(* Logix 5000 project; controller Receptivo vendor 1 type 14 code 106 rev 30.11; software revision 30.00; part 9 of 10 *)
(* tags used below, declared in another part *)
   Command_Status : DINT;
   Gway_Error : BOOL;
   GWay_Heartbeat : DINT;
   Gway_Status : DINT;
   ons_tare_station_3 : BOOL;
   ons_wpm3 : BOOL;
   ons_wpm4 : BOOL;
   Timer_Gway_Hearbeat : TIMER[4];
   Timer_Tare_Station_3 : TIMER;
   Timer_Tare_Station_3_aux : BOOL;
   Timer_Tare_Station_4 : TIMER;
   Timer_Tare_Station_4_aux : BOOL;
   Timer_WPM3_Heartbeat : TIMER[8];
   Timer_WPM4_Heartbeat : TIMER[8];
   WPM_3_COUNT_ANTERIOR : DINT;
   WPM_4_COUNT_ANTERIOR : DINT;
   ACTIVE_SLOT : DINT[10];
   CAJAS_1 : DINT;
   CAJAS_2 : DINT;
   CAJAS_3 : DINT;
   CAJAS_4 : DINT;
   CHASSIS_LAST : DINT;
   Diff_Peso_1 : DINT;
   Diff_Peso_2 : DINT;
   Diff_Peso_3 : DINT;
   Diff_Peso_4 : DINT;
   FORCE_STATUS : DINT;
   KEY_SWITCH_RUN : BOOL;
   MODULE_FAULT_STATUS : DINT[10];
   Num_Cajas_Reales_1 : DINT;
   Num_Cajas_Reales_2 : DINT;
   Num_Cajas_Reales_3 : DINT;
   Num_Cajas_Reales_4 : DINT;
   ons_tare_station_4 : BOOL;
   PB_Tare_Station_3 : BOOL;
   PB_Tare_Station_4 : BOOL;
   Peso_OK_Estacion_1 : BOOL;
   Peso_OK_Estacion_2 : BOOL;
   Peso_OK_Estacion_3 : BOOL;
   Peso_OK_Estacion_4 : BOOL;
   PESO_REAL_1 : DINT;
   PESO_REAL_2 : DINT;
   PESO_REAL_3 : DINT;
   PESO_REAL_4 : DINT;
   PESO_TEORICO_1 : DINT;
   PESO_TEORICO_2 : DINT;
   PESO_TEORICO_3 : DINT;
   PESO_TEORICO_4 : DINT;
   Porcentaje_Peso_1 : REAL;
   Porcentaje_Peso_2 : REAL;
   Porcentaje_Peso_3 : REAL;
   Porcentaje_Peso_4 : REAL;
   Producto1 : UDT_Inventario;
   Producto2 : UDT_Inventario;
   Producto3 : UDT_Inventario;
   Producto4 : UDT_Inventario;
   Station3_Tare_OK : BOOL;
   Station4_Tare_OK : BOOL;
   SYSTEM_ALARMS : DINT[10];
   Tara_1 : DINT;
   Tara_2 : DINT;
   Tara_3 : DINT;
   Tara_4 : DINT;
   Tara_Fecha_Estacion_3 : Hora_y_Fecha;
   Tara_Fecha_Estacion_4 : Hora_y_Fecha;
   Tare_Station_1_Write : DINT;
   Tare_Station_2_Write : DINT;
   Tare_Station_3_Write : DINT;
   Tare_Station_4_Write : DINT;
   WPM1_Heartbeat_Error : BOOL;
   WPM2_Heartbeat_Error : BOOL;
   WPM3_Heartbeat : DINT;
   WPM3_Heartbeat_Error : BOOL;
   WPM3_Status : WPM_Status;
   WPM4_Heartbeat : DINT;
   WPM4_Heartbeat_Error : BOOL;
   WPM4_Status : WPM_Status;
   WPM_3_Selected : DINT;
   WPM_3_Status_Aux : DINT;
   WPM_4_Selected : DINT;
   WPM_4_Status_Aux : DINT;
   Zero : DINT;
(* Pesaje, continued *)

ROUTINE Control_Pesaje_3   (* ladder *)
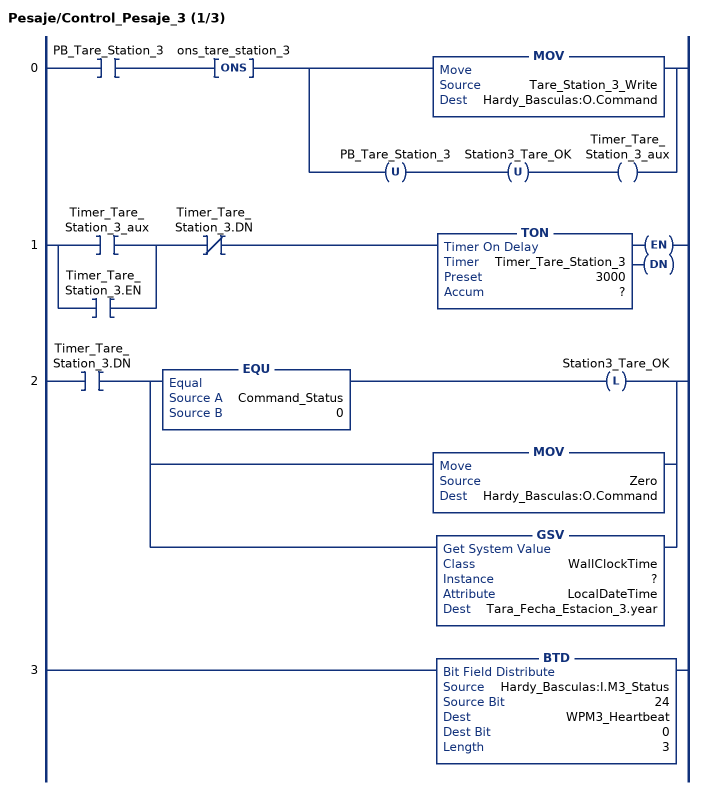
   0: XIC(PB_Tare_Station_3)ONS(ons_tare_station_3)[MOV(Tare_Station_3_Write,Hardy_Basculas:O.Command) ,OTU(PB_Tare_Station_3) OTU(Station3_Tare_OK) OTE(Timer_Tare_Station_3_aux) ];
   1: [XIC(Timer_Tare_Station_3_aux) ,XIC(Timer_Tare_Station_3.EN) ]XIO(Timer_Tare_Station_3.DN)TON(Timer_Tare_Station_3,?,?);
   2: XIC(Timer_Tare_Station_3.DN)[EQU(Command_Status,0) OTL(Station3_Tare_OK) ,MOV(Zero,Hardy_Basculas:O.Command) ,GSV(WallClockTime,?,LocalDateTime,Tara_Fecha_Estacion_3.year) ];
   3: BTD(Hardy_Basculas:I.M3_Status,24,WPM3_Heartbeat,0,3);
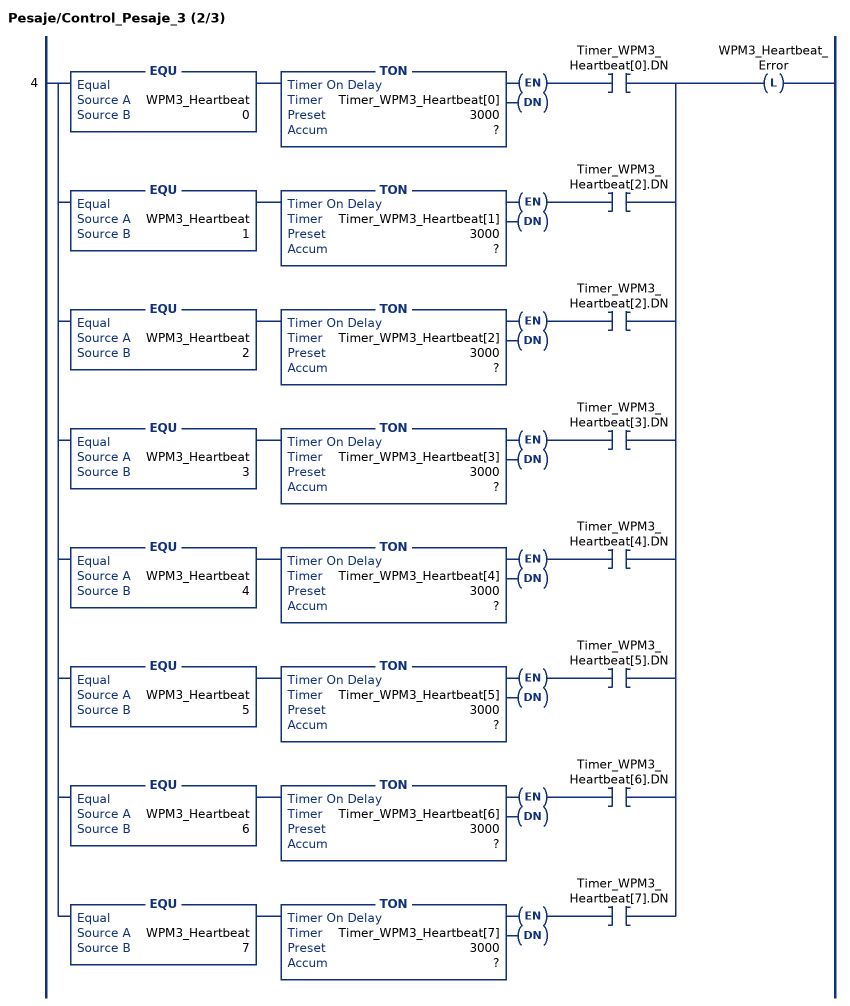
   4: [EQU(WPM3_Heartbeat,0) TON(Timer_WPM3_Heartbeat[0],?,?) XIC(Timer_WPM3_Heartbeat[0].DN) ,EQU(WPM3_Heartbeat,1) TON(Timer_WPM3_Heartbeat[1],?,?) XIC(Timer_WPM3_Heartbeat[2].DN) ,EQU(WPM3_Heartbeat,2) TON(Timer_WPM3_Heartbeat[2],?,?) XIC(Timer_WPM3_Heartbeat[2].DN) ,EQU(WPM3_Heartbeat,3) TON(Timer_WPM3_Heartbeat[3],?,?) XIC(Timer_WPM3_Heartbeat[3].DN) ,EQU(WPM3_Heartbeat,4) TON(Timer_WPM3_Heartbeat[4],?,?) XIC(Timer_WPM3_Heartbeat[4].DN) ,EQU(WPM3_Heartbeat,5) TON(Timer_WPM3_Heartbeat[5],?,?) XIC(Timer_WPM3_Heartbeat[5].DN) ,EQU(WPM3_Heartbeat,6) TON(Timer_WPM3_Heartbeat[6],?,?) XIC(Timer_WPM3_Heartbeat[6].DN) ,EQU(WPM3_Heartbeat,7) TON(Timer_WPM3_Heartbeat[7],?,?) XIC(Timer_WPM3_Heartbeat[7].DN) ]OTL(WPM3_Heartbeat_Error);
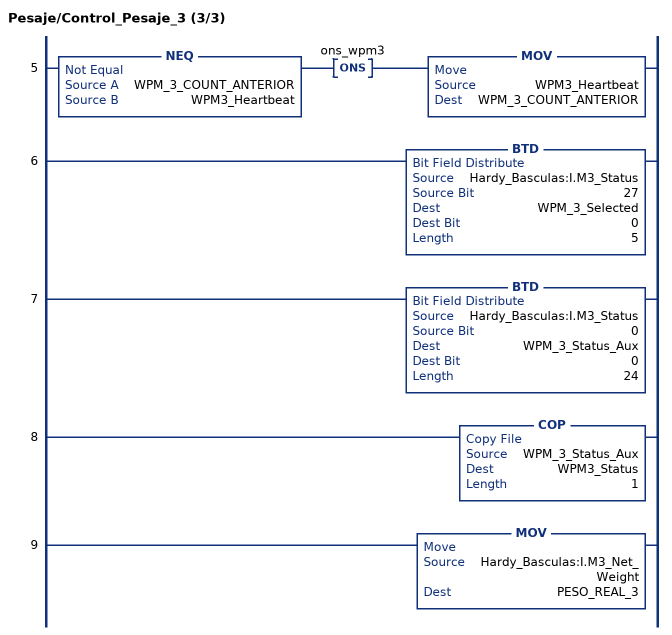
   5: NEQ(WPM_3_COUNT_ANTERIOR,WPM3_Heartbeat)ONS(ons_wpm3)MOV(WPM3_Heartbeat,WPM_3_COUNT_ANTERIOR);
   6: BTD(Hardy_Basculas:I.M3_Status,27,WPM_3_Selected,0,5);
   7: BTD(Hardy_Basculas:I.M3_Status,0,WPM_3_Status_Aux,0,24);
   8: COP(WPM_3_Status_Aux,WPM3_Status,1);
   9: MOV(Hardy_Basculas:I.M3_Net_Weight,PESO_REAL_3);
END_ROUTINE

ROUTINE Control_Pesaje_4   (* ladder *)
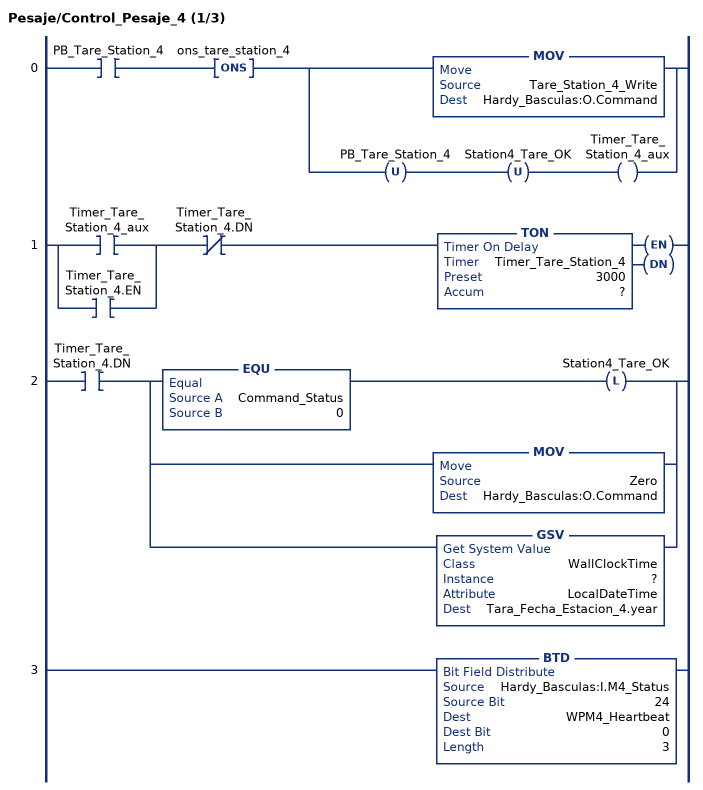
   0: XIC(PB_Tare_Station_4)ONS(ons_tare_station_4)[MOV(Tare_Station_4_Write,Hardy_Basculas:O.Command) ,OTU(PB_Tare_Station_4) OTU(Station4_Tare_OK) OTE(Timer_Tare_Station_4_aux) ];
   1: [XIC(Timer_Tare_Station_4_aux) ,XIC(Timer_Tare_Station_4.EN) ]XIO(Timer_Tare_Station_4.DN)TON(Timer_Tare_Station_4,?,?);
   2: XIC(Timer_Tare_Station_4.DN)[EQU(Command_Status,0) OTL(Station4_Tare_OK) ,MOV(Zero,Hardy_Basculas:O.Command) ,GSV(WallClockTime,?,LocalDateTime,Tara_Fecha_Estacion_4.year) ];
   3: BTD(Hardy_Basculas:I.M4_Status,24,WPM4_Heartbeat,0,3);
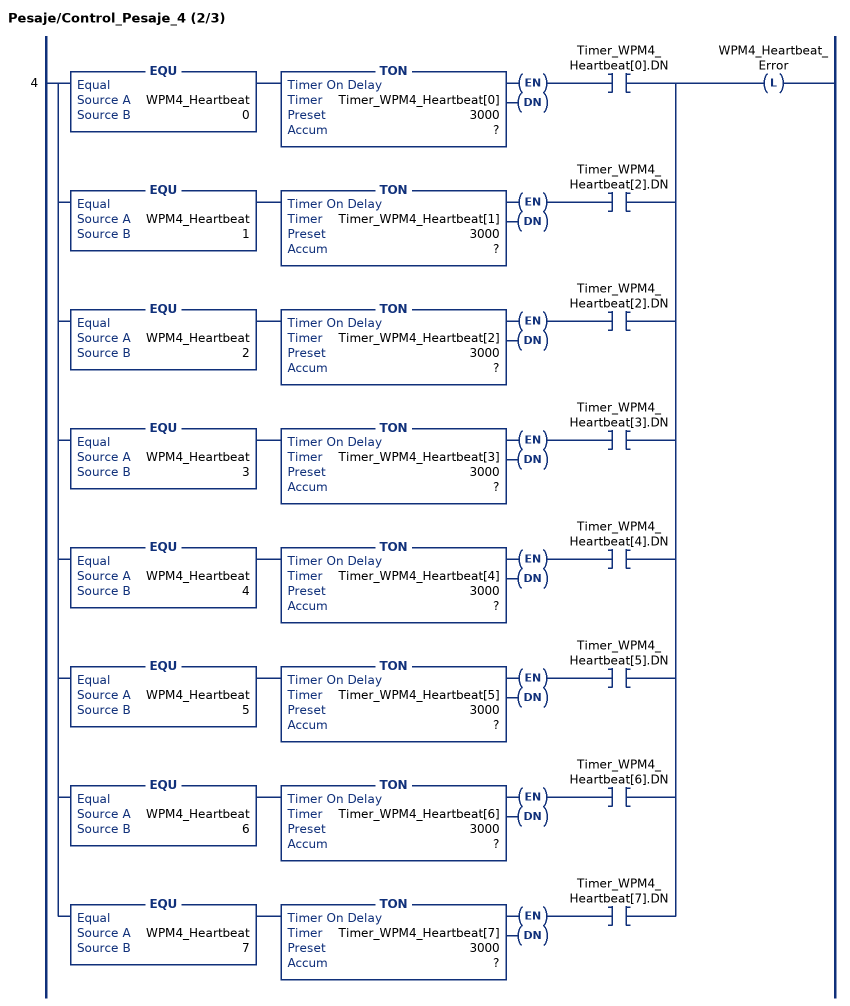
   4: [EQU(WPM4_Heartbeat,0) TON(Timer_WPM4_Heartbeat[0],?,?) XIC(Timer_WPM4_Heartbeat[0].DN) ,EQU(WPM4_Heartbeat,1) TON(Timer_WPM4_Heartbeat[1],?,?) XIC(Timer_WPM4_Heartbeat[2].DN) ,EQU(WPM4_Heartbeat,2) TON(Timer_WPM4_Heartbeat[2],?,?) XIC(Timer_WPM4_Heartbeat[2].DN) ,EQU(WPM4_Heartbeat,3) TON(Timer_WPM4_Heartbeat[3],?,?) XIC(Timer_WPM4_Heartbeat[3].DN) ,EQU(WPM4_Heartbeat,4) TON(Timer_WPM4_Heartbeat[4],?,?) XIC(Timer_WPM4_Heartbeat[4].DN) ,EQU(WPM4_Heartbeat,5) TON(Timer_WPM4_Heartbeat[5],?,?) XIC(Timer_WPM4_Heartbeat[5].DN) ,EQU(WPM4_Heartbeat,6) TON(Timer_WPM4_Heartbeat[6],?,?) XIC(Timer_WPM4_Heartbeat[6].DN) ,EQU(WPM4_Heartbeat,7) TON(Timer_WPM4_Heartbeat[7],?,?) XIC(Timer_WPM4_Heartbeat[7].DN) ]OTL(WPM4_Heartbeat_Error);
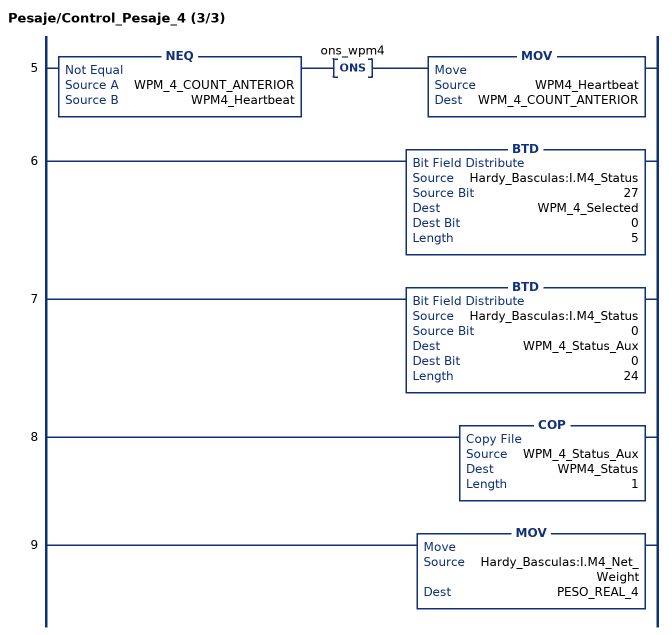
   5: NEQ(WPM_4_COUNT_ANTERIOR,WPM4_Heartbeat)ONS(ons_wpm4)MOV(WPM4_Heartbeat,WPM_4_COUNT_ANTERIOR);
   6: BTD(Hardy_Basculas:I.M4_Status,27,WPM_4_Selected,0,5);
   7: BTD(Hardy_Basculas:I.M4_Status,0,WPM_4_Status_Aux,0,24);
   8: COP(WPM_4_Status_Aux,WPM4_Status,1);
   9: MOV(Hardy_Basculas:I.M4_Net_Weight,PESO_REAL_4);
END_ROUTINE

ROUTINE Pesaje_Principal   (* ladder *)
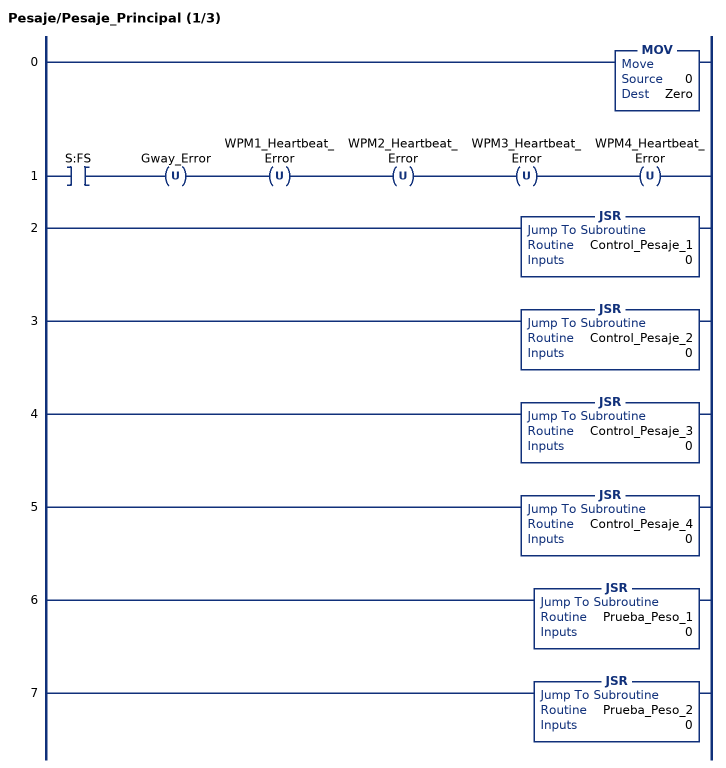
   0: MOV(0,Zero);
   1: XIC(S:FS)OTU(Gway_Error)OTU(WPM1_Heartbeat_Error)OTU(WPM2_Heartbeat_Error)OTU(WPM3_Heartbeat_Error)OTU(WPM4_Heartbeat_Error);
   2: JSR(Control_Pesaje_1,0);
   3: JSR(Control_Pesaje_2,0);
   4: JSR(Control_Pesaje_3,0);
   5: JSR(Control_Pesaje_4,0);
   6: JSR(Prueba_Peso_1,0);
   7: JSR(Prueba_Peso_2,0);
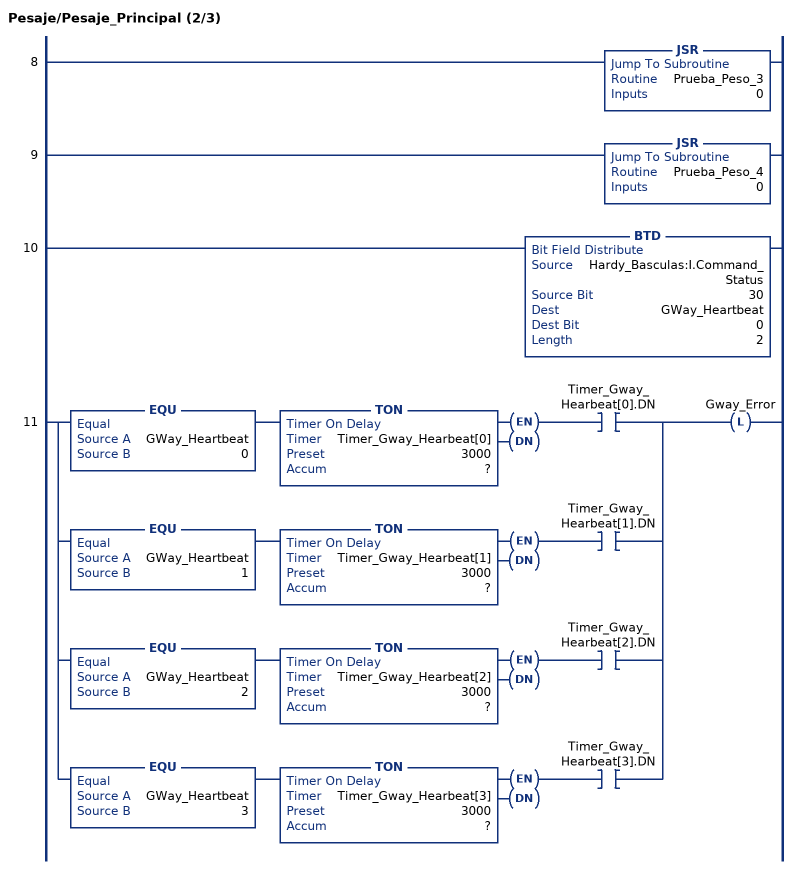
   8: JSR(Prueba_Peso_3,0);
   9: JSR(Prueba_Peso_4,0);
   10: BTD(Hardy_Basculas:I.Command_Status,30,GWay_Heartbeat,0,2);
   11: [EQU(GWay_Heartbeat,0) TON(Timer_Gway_Hearbeat[0],?,?) XIC(Timer_Gway_Hearbeat[0].DN) ,EQU(GWay_Heartbeat,1) TON(Timer_Gway_Hearbeat[1],?,?) XIC(Timer_Gway_Hearbeat[1].DN) ,EQU(GWay_Heartbeat,2) TON(Timer_Gway_Hearbeat[2],?,?) XIC(Timer_Gway_Hearbeat[2].DN) ,EQU(GWay_Heartbeat,3) TON(Timer_Gway_Hearbeat[3],?,?) XIC(Timer_Gway_Hearbeat[3].DN) ]OTL(Gway_Error);
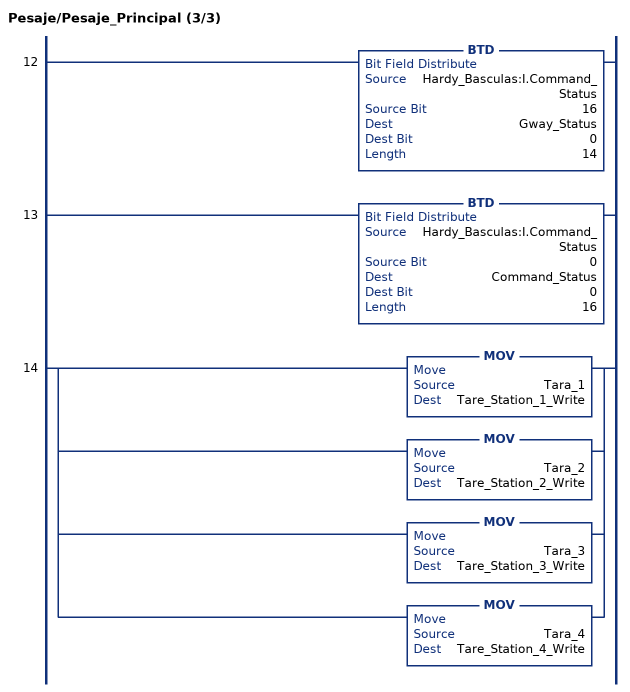
   12: BTD(Hardy_Basculas:I.Command_Status,16,Gway_Status,0,14);
   13: BTD(Hardy_Basculas:I.Command_Status,0,Command_Status,0,16);
   14: [MOV(Tara_1,Tare_Station_1_Write) ,MOV(Tara_2,Tare_Station_2_Write) ,MOV(Tara_3,Tare_Station_3_Write) ,MOV(Tara_4,Tare_Station_4_Write) ];
END_ROUTINE

ROUTINE Prueba_Peso_1   (* ladder *)
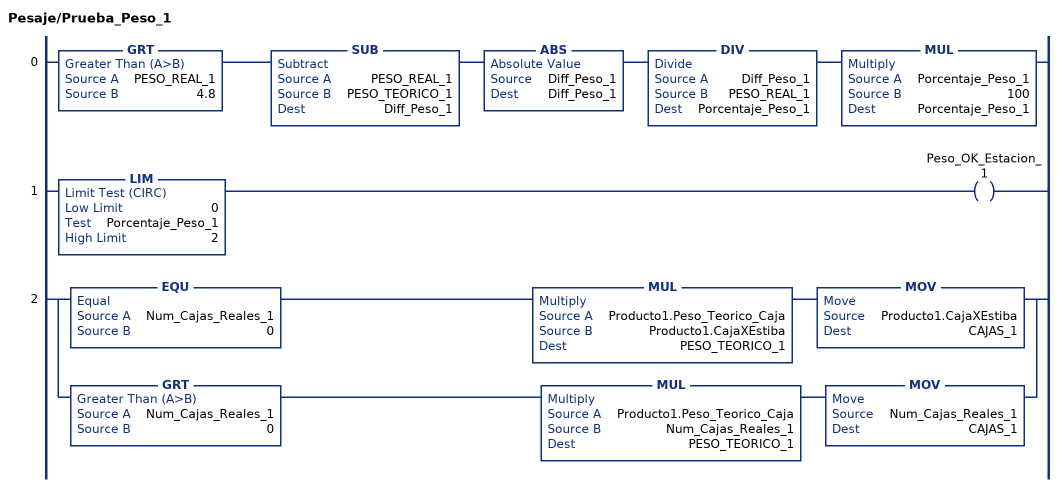
   0: GRT(PESO_REAL_1,4.8)SUB(PESO_REAL_1,PESO_TEORICO_1,Diff_Peso_1)ABS(Diff_Peso_1,Diff_Peso_1)DIV(Diff_Peso_1,PESO_REAL_1,Porcentaje_Peso_1)MUL(Porcentaje_Peso_1,100,Porcentaje_Peso_1);
   1: LIM(0,Porcentaje_Peso_1,2)OTE(Peso_OK_Estacion_1);
   2: [EQU(Num_Cajas_Reales_1,0) MUL(Producto1.Peso_Teorico_Caja,Producto1.CajaXEstiba,PESO_TEORICO_1) MOV(Producto1.CajaXEstiba,CAJAS_1) ,GRT(Num_Cajas_Reales_1,0) MUL(Producto1.Peso_Teorico_Caja,Num_Cajas_Reales_1,PESO_TEORICO_1) MOV(Num_Cajas_Reales_1,CAJAS_1) ];
END_ROUTINE

ROUTINE Prueba_Peso_2   (* ladder *)
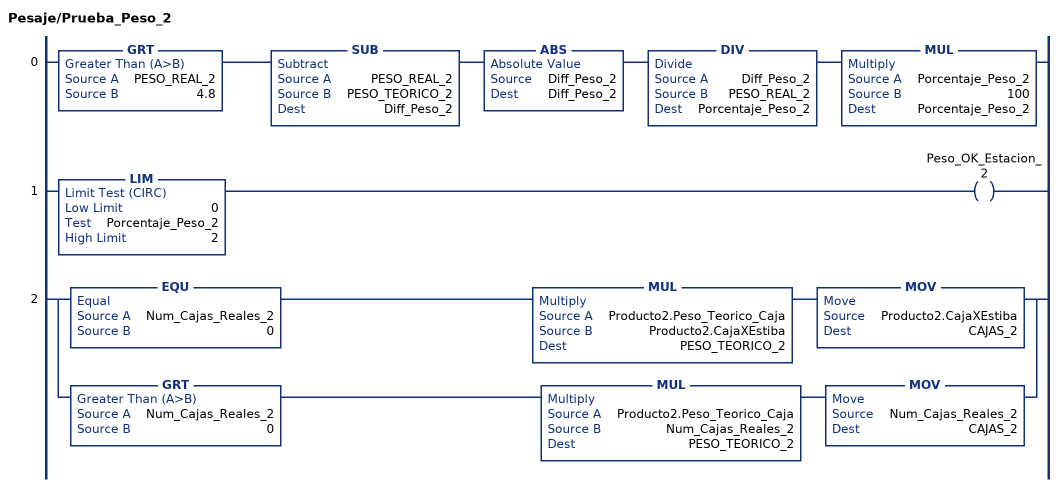
   0: GRT(PESO_REAL_2,4.8)SUB(PESO_REAL_2,PESO_TEORICO_2,Diff_Peso_2)ABS(Diff_Peso_2,Diff_Peso_2)DIV(Diff_Peso_2,PESO_REAL_2,Porcentaje_Peso_2)MUL(Porcentaje_Peso_2,100,Porcentaje_Peso_2);
   1: LIM(0,Porcentaje_Peso_2,2)OTE(Peso_OK_Estacion_2);
   2: [EQU(Num_Cajas_Reales_2,0) MUL(Producto2.Peso_Teorico_Caja,Producto2.CajaXEstiba,PESO_TEORICO_2) MOV(Producto2.CajaXEstiba,CAJAS_2) ,GRT(Num_Cajas_Reales_2,0) MUL(Producto2.Peso_Teorico_Caja,Num_Cajas_Reales_2,PESO_TEORICO_2) MOV(Num_Cajas_Reales_2,CAJAS_2) ];
END_ROUTINE

ROUTINE Prueba_Peso_3   (* ladder *)
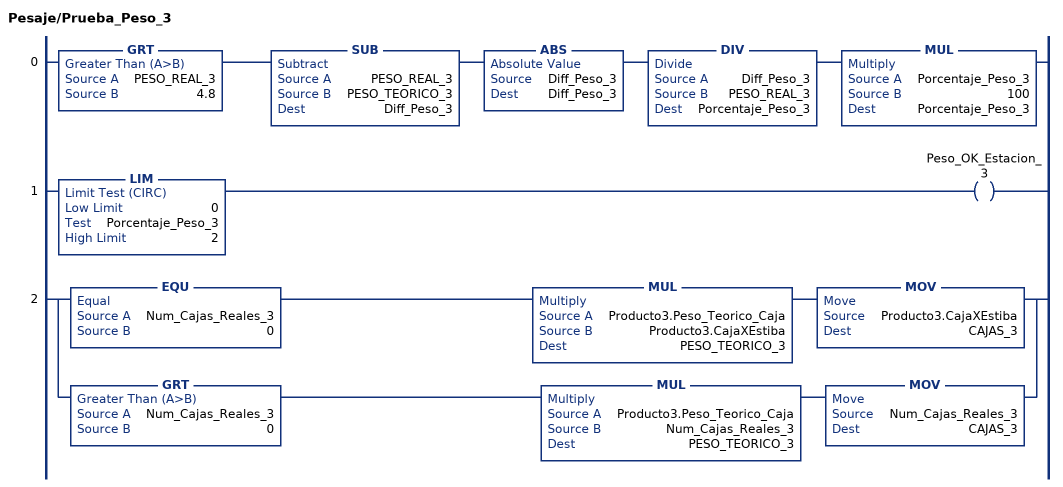
   0: GRT(PESO_REAL_3,4.8)SUB(PESO_REAL_3,PESO_TEORICO_3,Diff_Peso_3)ABS(Diff_Peso_3,Diff_Peso_3)DIV(Diff_Peso_3,PESO_REAL_3,Porcentaje_Peso_3)MUL(Porcentaje_Peso_3,100,Porcentaje_Peso_3);
   1: LIM(0,Porcentaje_Peso_3,2)OTE(Peso_OK_Estacion_3);
   2: [EQU(Num_Cajas_Reales_3,0) MUL(Producto3.Peso_Teorico_Caja,Producto3.CajaXEstiba,PESO_TEORICO_3) MOV(Producto3.CajaXEstiba,CAJAS_3) ,GRT(Num_Cajas_Reales_3,0) MUL(Producto3.Peso_Teorico_Caja,Num_Cajas_Reales_3,PESO_TEORICO_3) MOV(Num_Cajas_Reales_3,CAJAS_3) ];
END_ROUTINE

ROUTINE Prueba_Peso_4   (* ladder *)
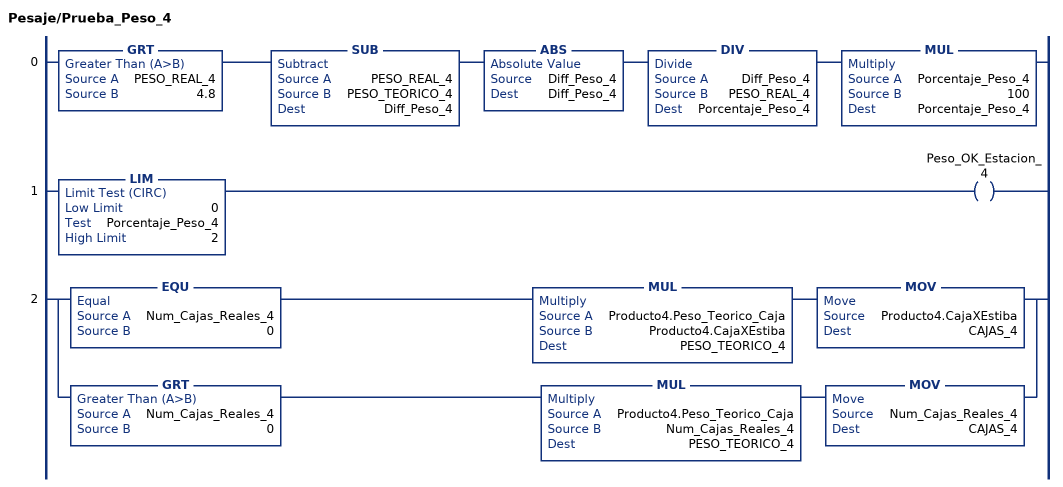
   0: GRT(PESO_REAL_4,4.8)SUB(PESO_REAL_4,PESO_TEORICO_4,Diff_Peso_4)ABS(Diff_Peso_4,Diff_Peso_4)DIV(Diff_Peso_4,PESO_REAL_4,Porcentaje_Peso_4)MUL(Porcentaje_Peso_4,100,Porcentaje_Peso_4);
   1: LIM(0,Porcentaje_Peso_4,2)OTE(Peso_OK_Estacion_4);
   2: [EQU(Num_Cajas_Reales_4,0) MUL(Producto4.Peso_Teorico_Caja,Producto4.CajaXEstiba,PESO_TEORICO_4) MOV(Producto4.CajaXEstiba,CAJAS_4) ,GRT(Num_Cajas_Reales_4,0) MUL(Producto4.Peso_Teorico_Caja,Num_Cajas_Reales_4,PESO_TEORICO_4) MOV(Num_Cajas_Reales_4,CAJAS_4) ];
END_ROUTINE
END_PROGRAM

PROGRAM SYSTEM_STATUS   (* main routine MAIN *)
VAR
   CHASSIS_CURRENT : INT := 1;
   CLOCK_SYNC : DINT[7] := ([5] := -1);
   CONTROLLER_STATUS : DINT := 12640;
   CPUdiag_AumaLOGO : INT := 8; {access Read Only}
   CPUdiag_FlashingGreen : BOOL; {access Read Only}
   CPUdiag_FlashingRed : BOOL; {access Read Only}
   CPUdiag_LEDStatus : DINT := 3; {access Read Only}
   CPUdiag_Major : MajorFaultBits;
   CPUdiag_MajorEvents : INT;
   CPUdiag_MajorFaultBits : DINT;
   CPUdiag_Minor : MinorFaultBits := (B_InstructionExecution := 1);
   CPUdiag_MinorEvents : INT := 21877;
   CPUdiag_MinorFaultBits : DINT := 16;
   CPUdiag_OneShot : BOOL[32]; {access None}
   CPUdiag_SolidGreen : BOOL := 1; {access Read Only}
   CPUdiag_StatusMasked : INT := 96;
   CPUdiag_StatusRaw : INT := 12640;
   CPUdiag_T : TIMER := (PRE := 300, ACC := 338); {access None}
   Dataman_Wireless_OK : BOOL;
   INDEX : INT := 16;
   IO_TREE_NO_OK : BOOL;
   IO_TREE_OK : DINT := 3;
   MINOR_FAULTS : DINT := 16;
   MODULE_MASK : DINT[10,17] := ([0,0] := 4096, [0,1] := 16384, [0,2] := 4096, [0,3] := 4096, [0,4] := 4096, [0,5] := 4096, [0,7] := 4096, [0,8] := 4096, [0,9] := 4096, [0,10] := 4096, [0,11] := 4096, [0,12] := 4096, [0,13] := 4096, [0,14] := 4096, [0,15] := 4096, [1,0] := 28672, [1,1] := 16384, [1,2] := 16384, [1,3] := 16384, [1,4] := 16384, [1,5] := 16384, [1,6] := 16384, [1,7] := 16384, [1,8] := 16384, [1,9] := 16384, [1,10] := 16384, [1,11] := 16384, [1,12] := 28672, [1,13] := 28672, [1,14] := 28672, [1,15] := 28672, [2,0] := 28672, [2,1] := 16384, [2,2] := 16384, [2,3] := 16384, [2,4] := 16384, [2,5] := 16384, [2,6] := 16384, [2,7] := 16384, [2,8] := 16384, [2,9] := 16384, [2,10] := 28672, [2,11] := 28672, [2,12] := 28672, [2,13] := 28672, [2,14] := 28672, [2,15] := 28672, [3,1] := 16384, [3,2] := 16384, [3,3] := 16384, [3,4] := 16384, [3,6] := 16384, [3,7] := 16384);
   MODULE_STATUS : DINT[10,17] := ([0,0] := 4096, [0,2] := 4096, [0,3] := 4096, [0,4] := 4096, [0,5] := 4096, [0,7] := 4096, [0,8] := 4096, [0,9] := 4096, [0,10] := 4096, [0,11] := 4096, [0,12] := 4096, [0,13] := 4096, [0,14] := 4096, [0,15] := 4096, [1,0] := 29184, [1,1] := 16384, [1,2] := 16384, [1,3] := 16384, [1,4] := 16384, [1,5] := 16384, [1,6] := 16384, [1,7] := 16384, [1,8] := 16384, [1,9] := 16384, [1,10] := 16897, [1,11] := 16897, [1,12] := 29184, [1,13] := 29184, [1,14] := 29184, [1,15] := 29184, [2,0] := 29184, [2,1] := 16897, [2,2] := 16897, [2,3] := 16897, [2,4] := 16897, [2,5] := 16897, [2,6] := 16897, [2,7] := 16897, [2,8] := 16897, [2,9] := 16897, [2,10] := 29184, [2,11] := 29184, [2,12] := 29184, [2,13] := 29184, [2,14] := 29184, [2,15] := 29184, [3,1] := 16897, [3,2] := 16897, [3,3] := 16897, [3,4] := 16897, [3,6] := 16897, [3,7] := 16897);
   Printer_Zebra_OK : BOOL := 1;
   Timer1 : TIMER := (PRE := 250, ACC := 67, EN := 1, TT := 1);
END_VAR

ROUTINE ALARMS   (* ladder *)
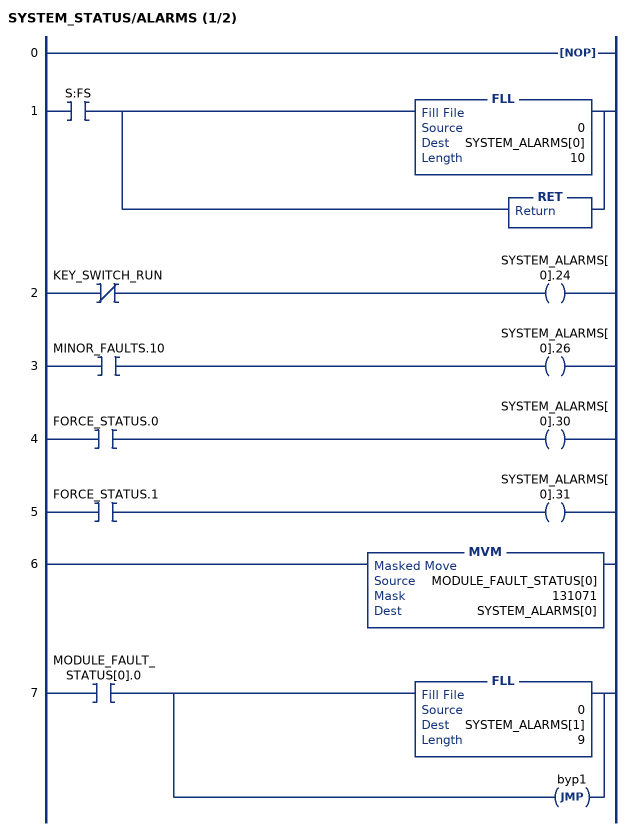
   0: NOP();
   1: XIC(S:FS)[FLL(0,SYSTEM_ALARMS[0],10) ,RET() ];
   2: XIO(KEY_SWITCH_RUN)OTE(SYSTEM_ALARMS[0].24);
   3: XIC(MINOR_FAULTS.10)OTE(SYSTEM_ALARMS[0].26);
   4: XIC(FORCE_STATUS.0)OTE(SYSTEM_ALARMS[0].30);
   5: XIC(FORCE_STATUS.1)OTE(SYSTEM_ALARMS[0].31);
   6: MVM(MODULE_FAULT_STATUS[0],131071,SYSTEM_ALARMS[0]);
   7: XIC(MODULE_FAULT_STATUS[0].0)[FLL(0,SYSTEM_ALARMS[1],9) ,JMP(byp1) ];
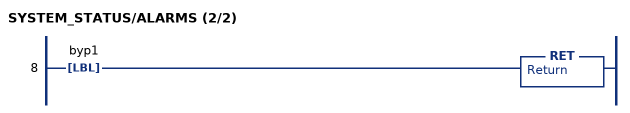
   8: LBL(byp1)RET();
END_ROUTINE

ROUTINE CONFIG   (* ladder *)
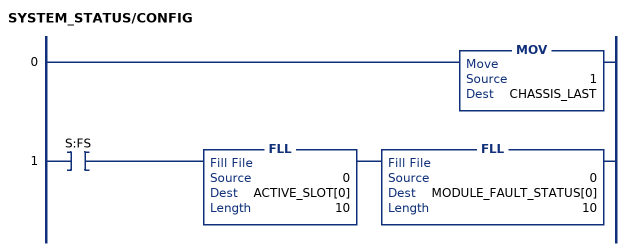
   0: MOV(1,CHASSIS_LAST);
   1: XIC(S:FS)FLL(0,ACTIVE_SLOT[0],10)FLL(0,MODULE_FAULT_STATUS[0],10);
END_ROUTINE

ROUTINE CONTROL   (* ladder *)
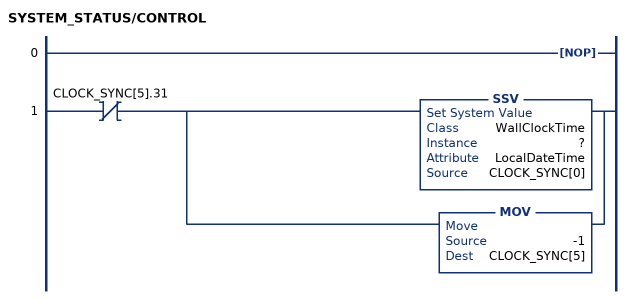
   0: NOP();
   1: XIO(CLOCK_SYNC[5].31)[SSV(WallClockTime,?,LocalDateTime,CLOCK_SYNC[0]) ,MOV(-1,CLOCK_SYNC[5]) ];
END_ROUTINE

ROUTINE CPU_STATUS_ON_HMI   (* ladder *)
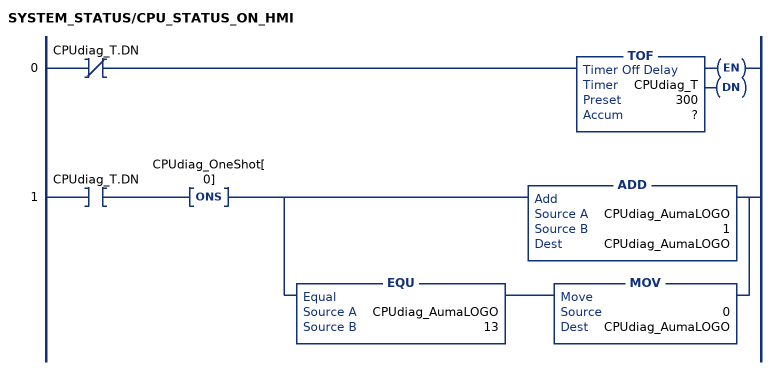
   0: XIO(CPUdiag_T.DN)TOF(CPUdiag_T,?,?);
   1: XIC(CPUdiag_T.DN)ONS(CPUdiag_OneShot[0])[ADD(CPUdiag_AumaLOGO,1,CPUdiag_AumaLOGO) ,EQU(CPUdiag_AumaLOGO,13) MOV(0,CPUdiag_AumaLOGO) ];
END_ROUTINE
